FUNCTION_BLOCK Consumer
  (* Standard: 61499-1 *)
  (* Version 1.0, 2026-07-29, Dimitrios Kalligaridis *)
  PACKAGE mypackage;
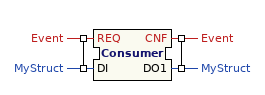
  EVENT_INPUT
    REQ WITH DI;
  END_EVENT
  EVENT_OUTPUT
    CNF WITH DO1;
  END_EVENT
  VAR_INPUT
    DI : mypackage::MyStruct;
  END_VAR
  VAR_OUTPUT
    DO1 : mypackage::MyStruct;
  END_VAR
  EC_STATES
    REQ : REQ -> CNF;
  END_STATES
  ALGORITHM REQ IN ST:

  END_ALGORITHM
END_FUNCTION_BLOCK
